FUNCTION_BLOCK Faults3
VAR_INPUT
	Execute : BOOL;
END_VAR
VAR_OUTPUT
END_VAR
VAR
END_VAR

IF Execute THEN
	Execute := FALSE;
END_IF

END_FUNCTION_BLOCK

(* stored: Version 1.1.0.1, ProductVersion 3.1.4024.11
   POU Faults3: Id {da3620e9-a87e-482d-bcc6-d5ae8b33990f}, SpecialFunc None *)
